// Mitsubishi GX Works2 project: 0702-6   PLC: Q02/Q02H

PROGRAM MAIN
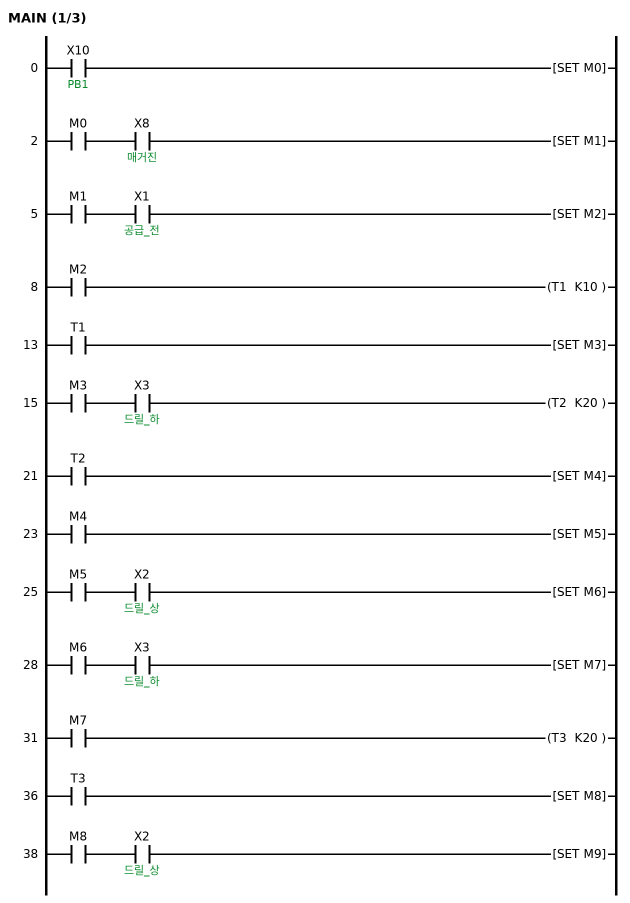
0     LD      X10  ; PB1
      SET     M0
2     LD      M0
      AND     X8  ; 매거진
      SET     M1
5     LD      M1
      AND     X1  ; 공급_전
      SET     M2
8     LD      M2
      OUT     T1 K10
13    LD      T1
      SET     M3
15    LD      M3
      AND     X3  ; 드릴_하
      OUT     T2 K20
21    LD      T2
      SET     M4
23    LD      M4
      SET     M5
25    LD      M5
      AND     X2  ; 드릴_상
      SET     M6
28    LD      M6
      AND     X3  ; 드릴_하
      SET     M7
31    LD      M7
      OUT     T3 K20
36    LD      T3
      SET     M8
38    LD      M8
      AND     X2  ; 드릴_상
      SET     M9
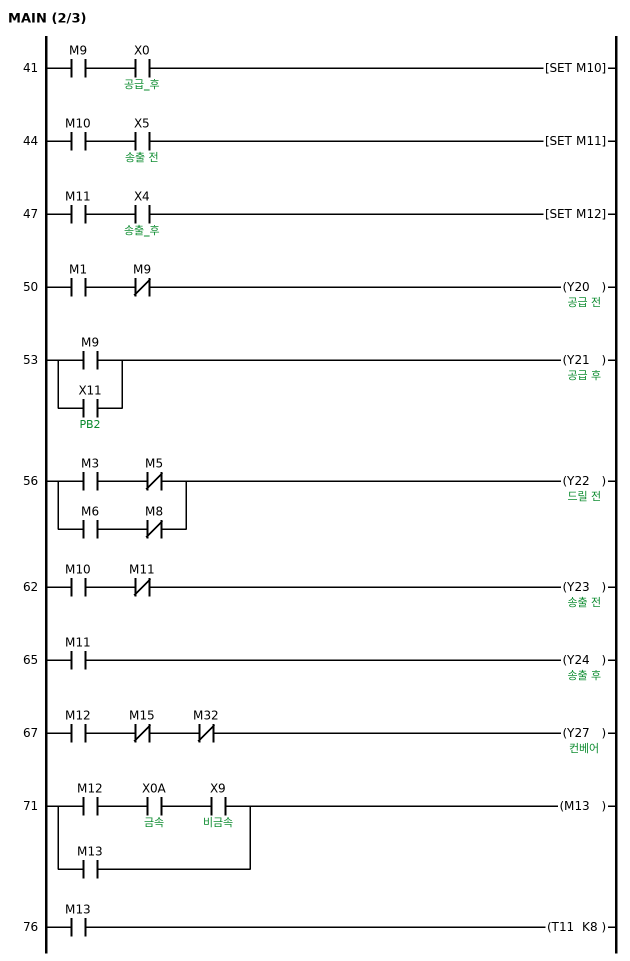
41    LD      M9
      AND     X0  ; 공급_후
      SET     M10
44    LD      M10
      AND     X5  ; 송출 전
      SET     M11
47    LD      M11
      AND     X4  ; 송출_후
      SET     M12
50    LD      M1
      ANI     M9
      OUT     Y20  ; 공급 전
53    LD      M9
      OR      X11  ; PB2
      OUT     Y21  ; 공급 후
56    LD      M3
      ANI     M5
      LD      M6
      ANI     M8
      ORB
      OUT     Y22  ; 드릴 전
62    LD      M10
      ANI     M11
      OUT     Y23  ; 송출 전
65    LD      M11
      OUT     Y24  ; 송출 후
67    LD      M12
      ANI     M15
      ANI     M32
      OUT     Y27  ; 컨베어
71    LD      M12
      AND     X0A  ; 금속
      AND     X9  ; 비금속
      OR      M13
      OUT     M13
76    LD      M13
      OUT     T11 K8
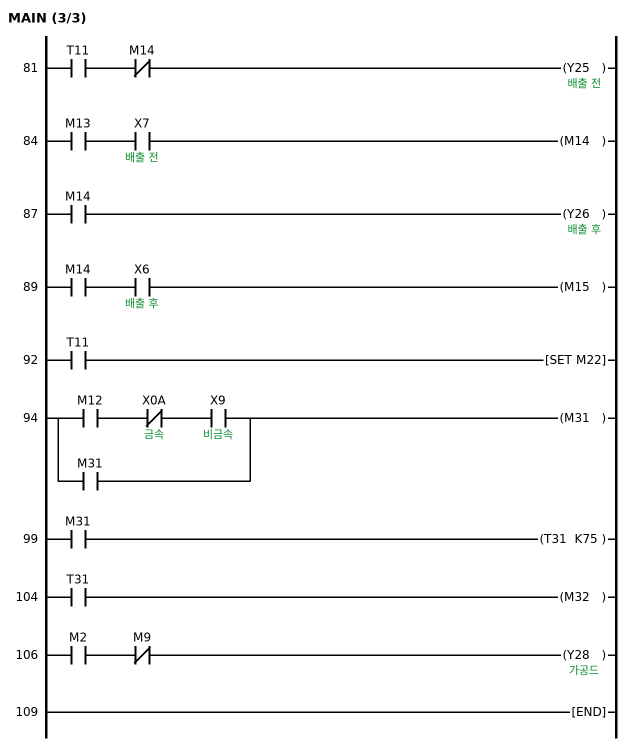
81    LD      T11
      ANI     M14
      OUT     Y25  ; 배출 전
84    LD      M13
      AND     X7  ; 배출 전
      OUT     M14
87    LD      M14
      OUT     Y26  ; 배출 후
89    LD      M14
      AND     X6  ; 배출 후
      OUT     M15
92    LD      T11
      SET     M22
94    LD      M12
      ANI     X0A  ; 금속
      AND     X9  ; 비금속
      OR      M31
      OUT     M31
99    LD      M31
      OUT     T31 K75
104   LD      T31
      OUT     M32
106   LD      M2
      ANI     M9
      OUT     Y28  ; 가공드
109   END
END_PROGRAM

// device comments not shown above
X12  ; PB3
Y29  ; 적색
Y2A  ; 황색
Y2B  ; 녹색
